(*udt (user defined type) of Graco Profibus Based Stud:
	auth.  Sodecia GTAC; 
	May 2013; version 1.0
	July 2020 Updated for new Graco GSD - j.vandongen
	*)

TYPE udt_Graco_Input :
	STRUCT
		(*Status Of Profibus Slave*)
		Inputs:udt_ProfiNode_Status;

		(*Input Bytes*)
		Byte0: BYTE;
		Byte1: BYTE;
		Byte2: BYTE;
		Byte3: BYTE;
		Byte4: BYTE;
		Byte5: BYTE;
		Byte6: BYTE;
		Byte7: BYTE;
		Byte8: BYTE;
		Byte9: BYTE;
		Byte10: BYTE;
		Byte11: BYTE;
		Byte12: BYTE;
		Byte13: BYTE;
		Byte14: BYTE;
		Byte15: BYTE;
		Byte16: BYTE;
		Byte17: BYTE;
		Byte18: BYTE;
		Byte19: BYTE;
		Byte20: BYTE;
		Byte21: BYTE;
		Byte22: BYTE;
		Byte23: BYTE;
		Byte24: BYTE;
		Byte25: BYTE;
		Byte26: BYTE;
		Byte27: BYTE;
		Byte28: BYTE;
		Byte29: BYTE;
		Byte30: BYTE;
		Byte31: BYTE;
		Byte32: BYTE;
		Byte33: BYTE;
		Byte34: BYTE;
		Byte35: BYTE;
		Byte36: BYTE;
		Byte37: BYTE;
		Byte38: BYTE;
		Byte39: BYTE;
		Byte40: BYTE;
		Byte41: BYTE;
		Byte42: BYTE;
		Byte43: BYTE;
		Byte44: BYTE;
		Byte45: BYTE;
		Byte46: BYTE;
		Byte47: BYTE;
		Byte48: BYTE;
		Byte49: BYTE;
		Byte50: BYTE;
		Byte51: BYTE;
		Byte52: BYTE;
		Byte53: BYTE;
		Byte54: BYTE;
		Byte55: BYTE;
		Byte56: BYTE;
		Byte57: BYTE;
		Byte58: BYTE;
		Byte59: BYTE;
		Byte60: BYTE;
		Byte61: BYTE;
		Byte62: BYTE;
		Byte63: BYTE;
		Byte64: BYTE;
		Byte65: BYTE;
		Byte66: BYTE;
		Byte67: BYTE;
		Byte68: BYTE;
		Byte69: BYTE;
		Byte70: BYTE;
		Byte71: BYTE;
		Byte72: BYTE;
		Byte73: BYTE;
		Byte74: BYTE;
		Byte75: BYTE;
		Byte76: BYTE;
		Byte77: BYTE;

	END_STRUCT
END_TYPE

(* stored: Version 1.1.0.1, ProductVersion 3.1.4024.5
   DUT udt_Graco_Input: Id {7b2ac0d6-6513-4988-a26a-442d10285716} *)
